Staubli VAL3: RefreshPage.pgx

program RefreshPage()
begin
  //
  gotoxy(1,1)
  put("--操作信息--")
  if !bPause
    gotoxy(1,13)
    put("暂停")
  else
    gotoxy(1,13)
    put("继续")
  endIf

  gotoxy(6,13)
  put("停止")
end
